// Mitsubishi GX Works2 project: abb_project_plc_135   PLC: Q03UDV

// global labels: Global1
VAR_GLOBAL
  공급후진리드 AT X20 : BOOL;
  공급전진리드 AT X21 : BOOL;
  매거진센서 AT X22 : BOOL;
  고주파센서 AT X23 : BOOL;
  용량형센서 AT X24 : BOOL;
  근접포토센서 AT X25 : BOOL;
  그리퍼온리드 AT X27 : BOOL;
  그리퍼오프리드 AT X28 : BOOL;
  물품도착포토 AT X29 : BOOL;
  TG1 AT X2A : BOOL;
  TG2 AT X2B : BOOL;
  TG3 AT X2C : BOOL;
  PB4 AT X2D : BOOL;
  PB5 AT X2E : BOOL;
  창고1 AT X30 : BOOL;
  창고2 AT X31 : BOOL;
  창고3 AT X32 : BOOL;
  창고4 AT X33 : BOOL;
  창고5 AT X34 : BOOL;
  창고6 AT X35 : BOOL;
  창고7 AT X36 : BOOL;
  창고8 AT X37 : BOOL;
  창고9 AT X38 : BOOL;
  도어센서 AT X39 : BOOL;
  압력센서 AT X3A : BOOL;
  공급전솔 AT Y40 : BOOL;
  공급후솔 AT Y41 : BOOL;
  그리퍼온솔 AT Y42 : BOOL;
  그리퍼오프솔 AT Y43 : BOOL;
  경광녹색 AT Y44 : BOOL;
  경광황색 AT Y45 : BOOL;
  경광적색 AT Y46 : BOOL;
  부저 AT Y47 : BOOL;
  컨베이어 AT Y48 : BOOL;
  램프1 AT Y4A : BOOL;
  램프2 AT Y4B : BOOL;
  램프3 AT Y4C : BOOL;
  램프4 AT Y4D : BOOL;
  램프5 AT Y4E : BOOL;
  R그립온명령 AT X1000 : BOOL;
  R그립오프명령 AT X1001 : BOOL;
  R_PLC시작 AT X1002 : BOOL;
  R_판별리셋 AT X1003 : BOOL;
  R재공급 AT X1004 : BOOL;
  R그립온센서 AT Y1000 : BOOL;
  R그립오프센서 AT Y1001 : BOOL;
  R물품없음 AT Y1002 : BOOL;
  R_금속 AT Y1003 : BOOL;
  R_검비금속 AT Y1004 : BOOL;
  R_흰비금속 AT Y1005 : BOOL;
  R물품도착 AT Y1006 : BOOL;
  R컨베이어 AT Y1007 : BOOL;
  R_재시작 AT Y1008 : BOOL;
  R_interrupt AT Y1009 : BOOL;
  R창고1 AT Y100A : BOOL;
  R창고2 AT Y100B : BOOL;
  R창고3 AT Y100C : BOOL;
  R창고4 AT Y100D : BOOL;
  R창고5 AT Y100E : BOOL;
  R창고6 AT Y100F : BOOL;
  R창고7 AT Y1010 : BOOL;
  R창고8 AT Y1011 : BOOL;
  R창고9 AT Y1012 : BOOL;
  R창고A AT Y1013 : BOOL;
  robot_reset AT X1005 : BOOL;
END_VAR

PROGRAM MAIN
VAR
  t물품없음 : TIMER;
  시작 : BOOL;
  공급전진 : BOOL;
  공급후진 : BOOL;
  재공급 : BOOL;
  컨구동 : BOOL;
  t컨정지지연 : TIMER;
  t컨베이어정지 : TIMER;
  용량형감지 : BOOL;
  고주파감지 : BOOL;
  근접포토감지 : BOOL;
  t감지지연 : TIMER;
  금속 : BOOL;
  비금속 : BOOL;
  흰플 : BOOL;
  검플 : BOOL;
  부저온 : BOOL;
  t창고7 : TIMER;
  t창고8 : TIMER;
  t창고9 : TIMER;
END_VAR
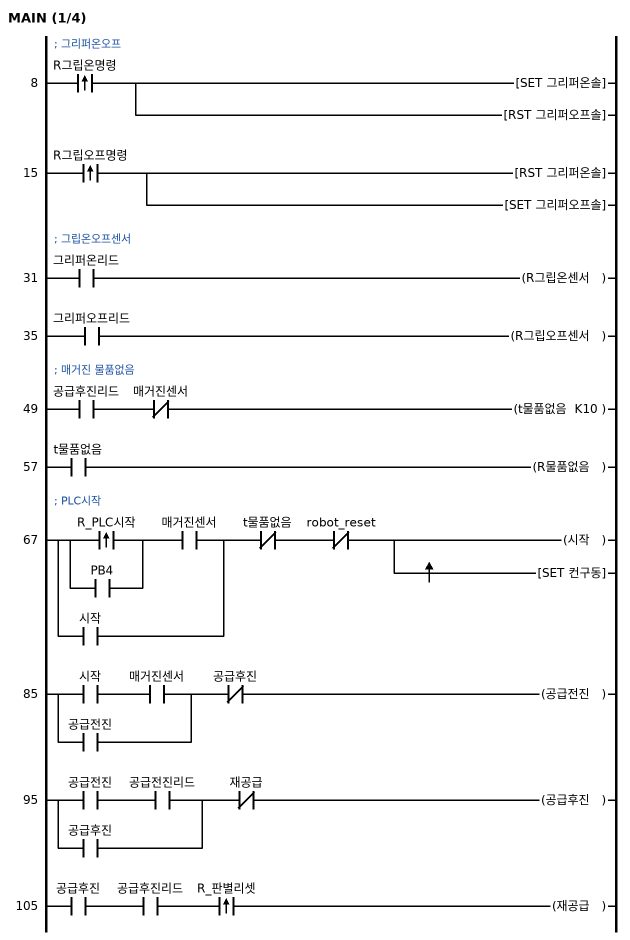
; 그리퍼온오프
8     LDP     R그립온명령
      SET     그리퍼온솔
      RST     그리퍼오프솔
15    LDP     R그립오프명령
      RST     그리퍼온솔
      SET     그리퍼오프솔
; 그립온오프센서
31    LD      그리퍼온리드
      OUT     R그립온센서
35    LD      그리퍼오프리드
      OUT     R그립오프센서
; 매거진 물품없음
49    LD      공급후진리드
      ANI     매거진센서
      OUT     t물품없음 K10
57    LD      t물품없음
      OUT     R물품없음
; PLC시작
67    LDP     R_PLC시작
      OR      PB4
      AND     매거진센서
      OR      시작
      ANI     t물품없음
      ANI     robot_reset
      OUT     시작
      MEP
      SET     컨구동
85    LD      시작
      AND     매거진센서
      OR      공급전진
      ANI     공급후진
      OUT     공급전진
95    LD      공급전진
      AND     공급전진리드
      OR      공급후진
      ANI     재공급
      OUT     공급후진
105   LD      공급후진
      AND     공급후진리드
      ANDP    R_판별리셋
      OUT     재공급
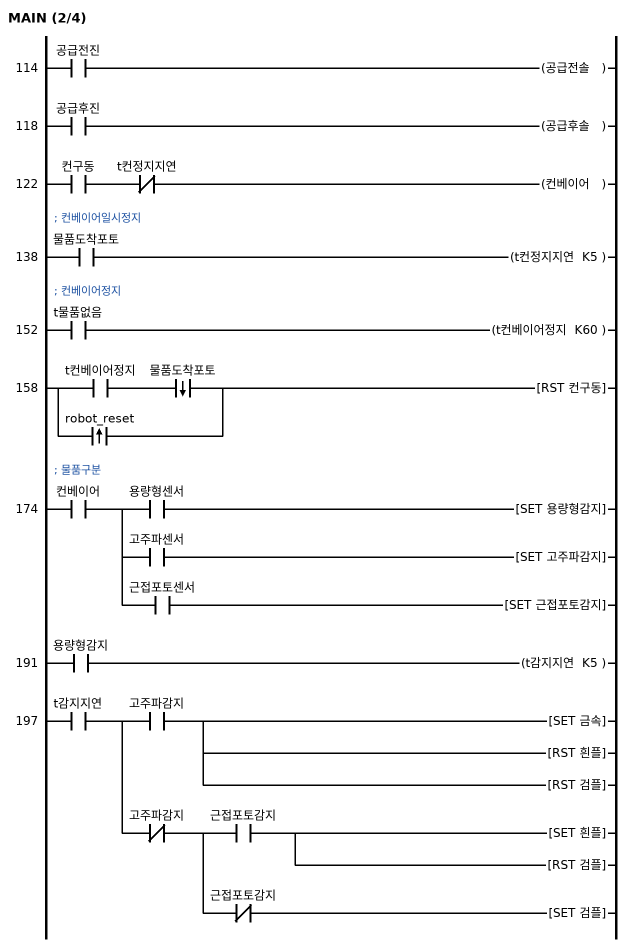
114   LD      공급전진
      OUT     공급전솔
118   LD      공급후진
      OUT     공급후솔
122   LD      컨구동
      ANI     t컨정지지연
      OUT     컨베이어
; 컨베이어일시정지
138   LD      물품도착포토
      OUT     t컨정지지연 K5
; 컨베이어정지
152   LD      t물품없음
      OUT     t컨베이어정지 K60
158   LD      t컨베이어정지
      ANDF    물품도착포토
      ORP     robot_reset
      RST     컨구동
; 물품구분
174   LD      컨베이어
      MPS
      AND     용량형센서
      SET     용량형감지
      MRD
      AND     고주파센서
      SET     고주파감지
      MPP
      AND     근접포토센서
      SET     근접포토감지
191   LD      용량형감지
      OUT     t감지지연 K5
197   LD      t감지지연
      MPS
      AND     고주파감지
      SET     금속
      RST     흰플
      RST     검플
      MPP
      ANI     고주파감지
      MPS
      AND     근접포토감지
      SET     흰플
      RST     검플
      MPP
      ANI     근접포토감지
      SET     검플
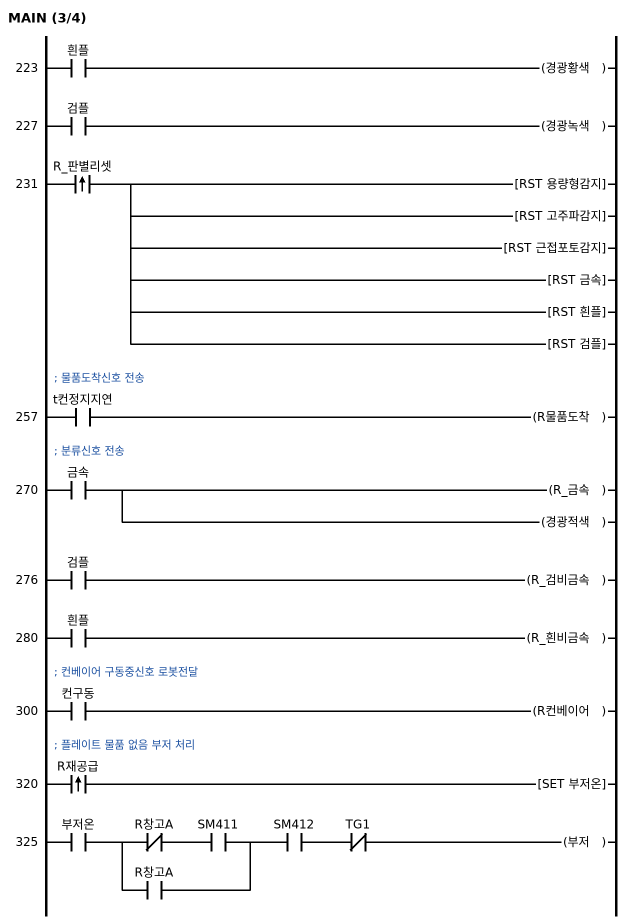
223   LD      흰플
      OUT     경광황색
227   LD      검플
      OUT     경광녹색
231   LDP     R_판별리셋
      RST     용량형감지
      RST     고주파감지
      RST     근접포토감지
      RST     금속
      RST     흰플
      RST     검플
; 물품도착신호 전송
257   LD      t컨정지지연
      OUT     R물품도착
; 분류신호 전송
270   LD      금속
      OUT     R_금속
      OUT     경광적색
276   LD      검플
      OUT     R_검비금속
280   LD      흰플
      OUT     R_흰비금속
; 컨베이어 구동중신호 로봇전달
300   LD      컨구동
      OUT     R컨베이어
; 플레이트 물품 없음 부저 처리
320   LDP     R재공급
      SET     부저온
325   LD      부저온
      LDI     R창고A
      AND     SM411
      OR      R창고A
      ANB
      AND     SM412
      ANI     TG1
      OUT     부저
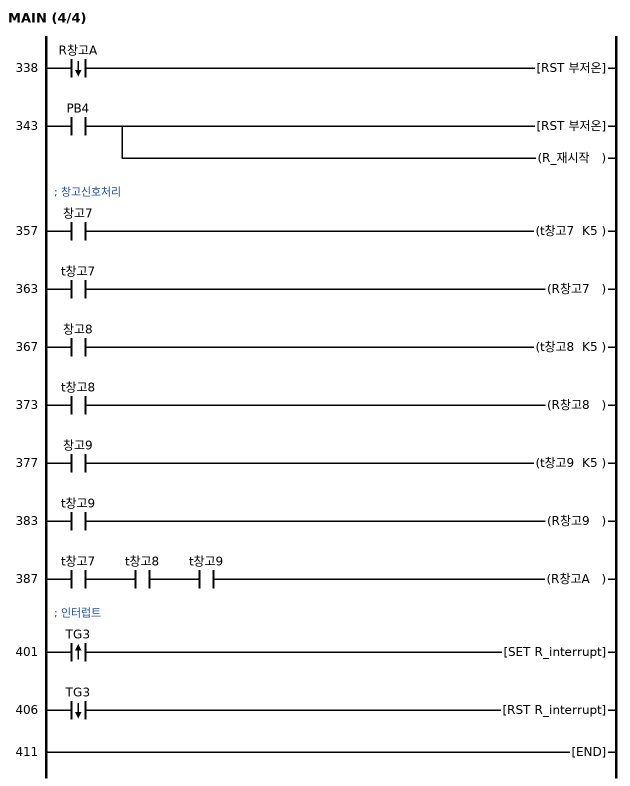
338   LDF     R창고A
      RST     부저온
343   LD      PB4
      RST     부저온
      OUT     R_재시작
; 창고신호처리
357   LD      창고7
      OUT     t창고7 K5
363   LD      t창고7
      OUT     R창고7
367   LD      창고8
      OUT     t창고8 K5
373   LD      t창고8
      OUT     R창고8
377   LD      창고9
      OUT     t창고9 K5
383   LD      t창고9
      OUT     R창고9
387   LD      t창고7
      AND     t창고8
      AND     t창고9
      OUT     R창고A
; 인터럽트
401   LDP     TG3
      SET     R_interrupt
406   LDF     TG3
      RST     R_interrupt
411   END
END_PROGRAM
